// TIA Portal V16 export
// export: Created 2021-11-12T13:31:11.9481413Z, ExportSetting WithDefaults, DisplayName Totally Integrated Automation Portal, DisplayVersion V16 Update 3, DisplayName TIA Portal Version Control Interface, DisplayVersion V16 Update 2, DisplayName TIA Portal Openness, DisplayVersion V16 Update 3, DisplayName SINAMICS Startdrive Advanced, DisplayVersion V16 Update 5, DisplayName SINAMICS Startdrive G130, G150, S120, S150, SINAMICS MV, S210, DisplayVersion V16 Update 5, DisplayName SINAMICS Startdrive G110M, G120, G120C, G120D, G120P, G115D, DisplayVersion V16 Update 5, DisplayName STEP 7 Professional, DisplayVersion V16 Update 3, DisplayName STEP 7 Safety, DisplayVersion V16, DisplayName WinCC UA Professional, DisplayVersion V16 Update 3
FUNCTION "Sfty_ProfiSafeCommIn" : Void   // FC23, F_LAD
{ S7_Optimized_Access := 'TRUE' }
VERSION : 0.1
// Wrintin Profisafe inputs into safety data block
// stored: AutoNumber true, IsIECCheckEnabled false, UDAEnableTagReadback false
BEGIN

REGION Network 1: *************** Robots section start ***************
END_REGION

REGION Network 2: 1R1+RC01
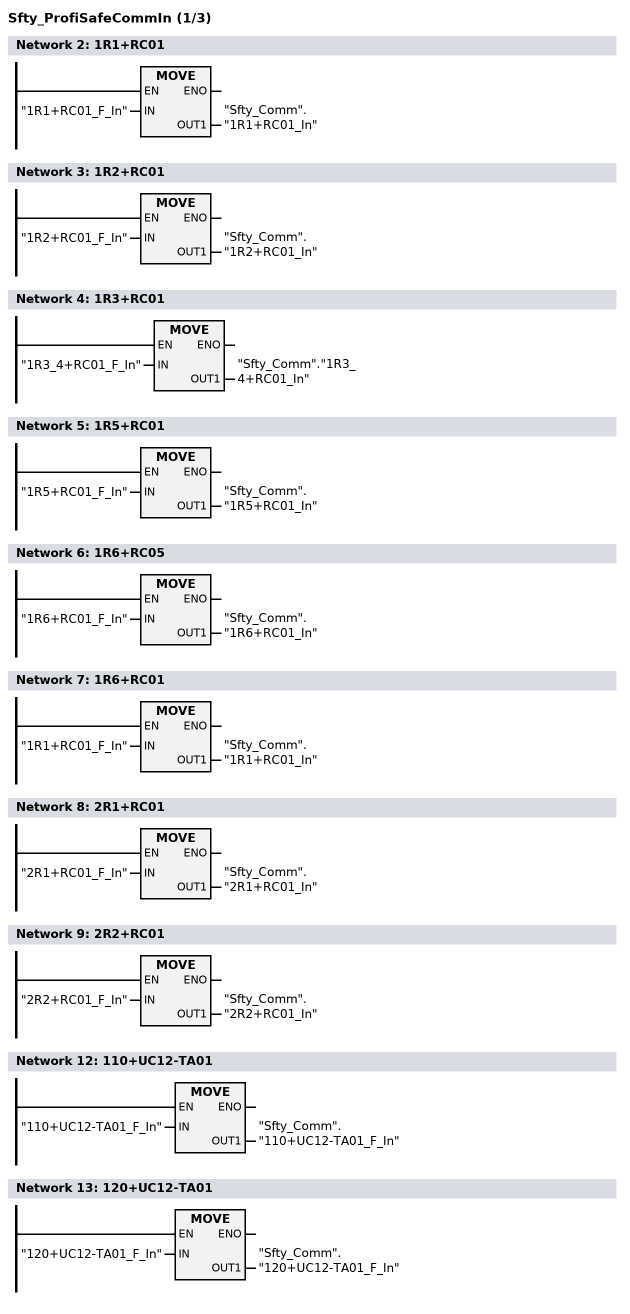
   RUNG wire#powerrail
      { S7_GenerateENO := "TRUE" } Move(in := "1R1+RC01_F_In", out1 => "Sfty_Comm"."1R1+RC01_In")
   END_RUNG
   // the same network as SCL:
   "Sfty_Comm"."1R1+RC01_In" := "1R1+RC01_F_In";
END_REGION

REGION Network 3: 1R2+RC01
   RUNG wire#powerrail
      { S7_GenerateENO := "TRUE" } Move(in := "1R2+RC01_F_In", out1 => "Sfty_Comm"."1R2+RC01_In")
   END_RUNG
   // the same network as SCL:
   "Sfty_Comm"."1R2+RC01_In" := "1R2+RC01_F_In";
END_REGION

REGION Network 4: 1R3+RC01
   RUNG wire#powerrail
      { S7_GenerateENO := "TRUE" } Move(in := "1R3_4+RC01_F_In", out1 => "Sfty_Comm"."1R3_4+RC01_In")
   END_RUNG
   // the same network as SCL:
   "Sfty_Comm"."1R3_4+RC01_In" := "1R3_4+RC01_F_In";
END_REGION

REGION Network 5: 1R5+RC01
   RUNG wire#powerrail
      { S7_GenerateENO := "TRUE" } Move(in := "1R5+RC01_F_In", out1 => "Sfty_Comm"."1R5+RC01_In")
   END_RUNG
   // the same network as SCL:
   "Sfty_Comm"."1R5+RC01_In" := "1R5+RC01_F_In";
END_REGION

REGION Network 6: 1R6+RC05
   RUNG wire#powerrail
      { S7_GenerateENO := "TRUE" } Move(in := "1R6+RC01_F_In", out1 => "Sfty_Comm"."1R6+RC01_In")
   END_RUNG
   // the same network as SCL:
   "Sfty_Comm"."1R6+RC01_In" := "1R6+RC01_F_In";
END_REGION

REGION Network 7: 1R6+RC01
   RUNG wire#powerrail
      { S7_GenerateENO := "TRUE" } Move(in := "1R1+RC01_F_In", out1 => "Sfty_Comm"."1R1+RC01_In")
   END_RUNG
   // the same network as SCL:
   "Sfty_Comm"."1R1+RC01_In" := "1R1+RC01_F_In";
END_REGION

REGION Network 8: 2R1+RC01
   RUNG wire#powerrail
      { S7_GenerateENO := "TRUE" } Move(in := "2R1+RC01_F_In", out1 => "Sfty_Comm"."2R1+RC01_In")
   END_RUNG
   // the same network as SCL:
   "Sfty_Comm"."2R1+RC01_In" := "2R1+RC01_F_In";
END_REGION

REGION Network 9: 2R2+RC01
   RUNG wire#powerrail
      { S7_GenerateENO := "TRUE" } Move(in := "2R2+RC01_F_In", out1 => "Sfty_Comm"."2R2+RC01_In")
   END_RUNG
   // the same network as SCL:
   "Sfty_Comm"."2R2+RC01_In" := "2R2+RC01_F_In";
END_REGION

REGION Network 10: *************** Robots section end ***************
END_REGION

REGION Network 11: *************** Inverters section start ***************
END_REGION

REGION Network 12: 110+UC12-TA01
   RUNG wire#powerrail
      { S7_GenerateENO := "TRUE" } Move(in := "110+UC12-TA01_F_In", out1 => "Sfty_Comm"."110+UC12-TA01_F_In")
   END_RUNG
   // the same network as SCL:
   "Sfty_Comm"."110+UC12-TA01_F_In" := "110+UC12-TA01_F_In";
END_REGION

REGION Network 13: 120+UC12-TA01
   RUNG wire#powerrail
      { S7_GenerateENO := "TRUE" } Move(in := "120+UC12-TA01_F_In", out1 => "Sfty_Comm"."120+UC12-TA01_F_In")
   END_RUNG
   // the same network as SCL:
   "Sfty_Comm"."120+UC12-TA01_F_In" := "120+UC12-TA01_F_In";
END_REGION

REGION Network 14: 210+UC12-TA01
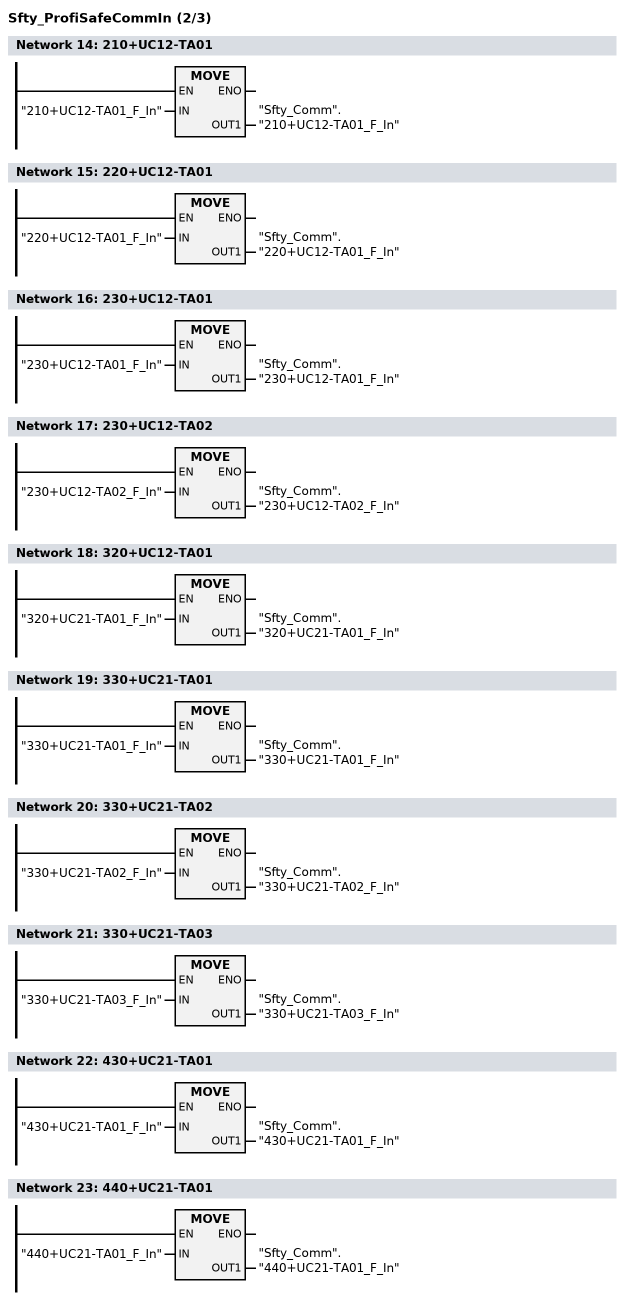
   RUNG wire#powerrail
      { S7_GenerateENO := "TRUE" } Move(in := "210+UC12-TA01_F_In", out1 => "Sfty_Comm"."210+UC12-TA01_F_In")
   END_RUNG
   // the same network as SCL:
   "Sfty_Comm"."210+UC12-TA01_F_In" := "210+UC12-TA01_F_In";
END_REGION

REGION Network 15: 220+UC12-TA01
   RUNG wire#powerrail
      { S7_GenerateENO := "TRUE" } Move(in := "220+UC12-TA01_F_In", out1 => "Sfty_Comm"."220+UC12-TA01_F_In")
   END_RUNG
   // the same network as SCL:
   "Sfty_Comm"."220+UC12-TA01_F_In" := "220+UC12-TA01_F_In";
END_REGION

REGION Network 16: 230+UC12-TA01
   RUNG wire#powerrail
      { S7_GenerateENO := "TRUE" } Move(in := "230+UC12-TA01_F_In", out1 => "Sfty_Comm"."230+UC12-TA01_F_In")
   END_RUNG
   // the same network as SCL:
   "Sfty_Comm"."230+UC12-TA01_F_In" := "230+UC12-TA01_F_In";
END_REGION

REGION Network 17: 230+UC12-TA02
   RUNG wire#powerrail
      { S7_GenerateENO := "TRUE" } Move(in := "230+UC12-TA02_F_In", out1 => "Sfty_Comm"."230+UC12-TA02_F_In")
   END_RUNG
   // the same network as SCL:
   "Sfty_Comm"."230+UC12-TA02_F_In" := "230+UC12-TA02_F_In";
END_REGION

REGION Network 18: 320+UC12-TA01
   RUNG wire#powerrail
      { S7_GenerateENO := "TRUE" } Move(in := "320+UC21-TA01_F_In", out1 => "Sfty_Comm"."320+UC21-TA01_F_In")
   END_RUNG
   // the same network as SCL:
   "Sfty_Comm"."320+UC21-TA01_F_In" := "320+UC21-TA01_F_In";
END_REGION

REGION Network 19: 330+UC21-TA01
   RUNG wire#powerrail
      { S7_GenerateENO := "TRUE" } Move(in := "330+UC21-TA01_F_In", out1 => "Sfty_Comm"."330+UC21-TA01_F_In")
   END_RUNG
   // the same network as SCL:
   "Sfty_Comm"."330+UC21-TA01_F_In" := "330+UC21-TA01_F_In";
END_REGION

REGION Network 20: 330+UC21-TA02
   RUNG wire#powerrail
      { S7_GenerateENO := "TRUE" } Move(in := "330+UC21-TA02_F_In", out1 => "Sfty_Comm"."330+UC21-TA02_F_In")
   END_RUNG
   // the same network as SCL:
   "Sfty_Comm"."330+UC21-TA02_F_In" := "330+UC21-TA02_F_In";
END_REGION

REGION Network 21: 330+UC21-TA03
   RUNG wire#powerrail
      { S7_GenerateENO := "TRUE" } Move(in := "330+UC21-TA03_F_In", out1 => "Sfty_Comm"."330+UC21-TA03_F_In")
   END_RUNG
   // the same network as SCL:
   "Sfty_Comm"."330+UC21-TA03_F_In" := "330+UC21-TA03_F_In";
END_REGION

REGION Network 22: 430+UC21-TA01
   RUNG wire#powerrail
      { S7_GenerateENO := "TRUE" } Move(in := "430+UC21-TA01_F_In", out1 => "Sfty_Comm"."430+UC21-TA01_F_In")
   END_RUNG
   // the same network as SCL:
   "Sfty_Comm"."430+UC21-TA01_F_In" := "430+UC21-TA01_F_In";
END_REGION

REGION Network 23: 440+UC21-TA01
   RUNG wire#powerrail
      { S7_GenerateENO := "TRUE" } Move(in := "440+UC21-TA01_F_In", out1 => "Sfty_Comm"."440+UC21-TA01_F_In")
   END_RUNG
   // the same network as SCL:
   "Sfty_Comm"."440+UC21-TA01_F_In" := "440+UC21-TA01_F_In";
END_REGION

REGION Network 24: 450+UC21-TA01
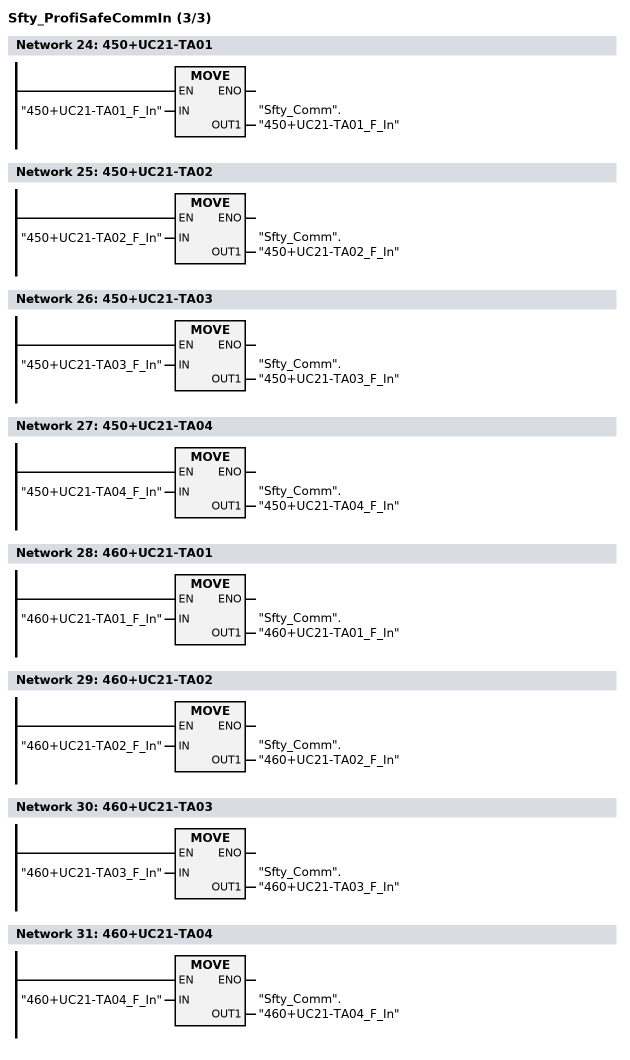
   RUNG wire#powerrail
      { S7_GenerateENO := "TRUE" } Move(in := "450+UC21-TA01_F_In", out1 => "Sfty_Comm"."450+UC21-TA01_F_In")
   END_RUNG
   // the same network as SCL:
   "Sfty_Comm"."450+UC21-TA01_F_In" := "450+UC21-TA01_F_In";
END_REGION

REGION Network 25: 450+UC21-TA02
   RUNG wire#powerrail
      { S7_GenerateENO := "TRUE" } Move(in := "450+UC21-TA02_F_In", out1 => "Sfty_Comm"."450+UC21-TA02_F_In")
   END_RUNG
   // the same network as SCL:
   "Sfty_Comm"."450+UC21-TA02_F_In" := "450+UC21-TA02_F_In";
END_REGION

REGION Network 26: 450+UC21-TA03
   RUNG wire#powerrail
      { S7_GenerateENO := "TRUE" } Move(in := "450+UC21-TA03_F_In", out1 => "Sfty_Comm"."450+UC21-TA03_F_In")
   END_RUNG
   // the same network as SCL:
   "Sfty_Comm"."450+UC21-TA03_F_In" := "450+UC21-TA03_F_In";
END_REGION

REGION Network 27: 450+UC21-TA04
   RUNG wire#powerrail
      { S7_GenerateENO := "TRUE" } Move(in := "450+UC21-TA04_F_In", out1 => "Sfty_Comm"."450+UC21-TA04_F_In")
   END_RUNG
   // the same network as SCL:
   "Sfty_Comm"."450+UC21-TA04_F_In" := "450+UC21-TA04_F_In";
END_REGION

REGION Network 28: 460+UC21-TA01
   RUNG wire#powerrail
      { S7_GenerateENO := "TRUE" } Move(in := "460+UC21-TA01_F_In", out1 => "Sfty_Comm"."460+UC21-TA01_F_In")
   END_RUNG
   // the same network as SCL:
   "Sfty_Comm"."460+UC21-TA01_F_In" := "460+UC21-TA01_F_In";
END_REGION

REGION Network 29: 460+UC21-TA02
   RUNG wire#powerrail
      { S7_GenerateENO := "TRUE" } Move(in := "460+UC21-TA02_F_In", out1 => "Sfty_Comm"."460+UC21-TA02_F_In")
   END_RUNG
   // the same network as SCL:
   "Sfty_Comm"."460+UC21-TA02_F_In" := "460+UC21-TA02_F_In";
END_REGION

REGION Network 30: 460+UC21-TA03
   RUNG wire#powerrail
      { S7_GenerateENO := "TRUE" } Move(in := "460+UC21-TA03_F_In", out1 => "Sfty_Comm"."460+UC21-TA03_F_In")
   END_RUNG
   // the same network as SCL:
   "Sfty_Comm"."460+UC21-TA03_F_In" := "460+UC21-TA03_F_In";
END_REGION

REGION Network 31: 460+UC21-TA04
   RUNG wire#powerrail
      { S7_GenerateENO := "TRUE" } Move(in := "460+UC21-TA04_F_In", out1 => "Sfty_Comm"."460+UC21-TA04_F_In")
   END_RUNG
   // the same network as SCL:
   "Sfty_Comm"."460+UC21-TA04_F_In" := "460+UC21-TA04_F_In";
END_REGION

REGION Network 32: *************** Inverters section start ***************
END_REGION
END_FUNCTION
